{attribute 'qualified_only'}
{attribute 'strict'}
TYPE E_BOHRER_STATES :
(
	eBereit := 0,
	eHerunterfahrend,
	eHochfahrend,
	eUnten,
	eOben,
	eFertig
);
END_TYPE

(* stored: Version 1.1.0.1, ProductVersion 3.1.4024.3
   DUT E_BOHRER_STATES: Id {752cddb8-db7f-4e28-b8f1-3a2f2368ecd8} *)
